FUNCTION_BLOCK MOTOR_TO_EVENTS (* Basic Function Block Type *)
  (* Standard: 61499-2 *)
  (* Version 0.3, 2009-09-15, JHC, Holobloc Inc, Changed transition priorities. *)
  (* Version 0.2, 2003-12-04, JHC, Rockwell Automation, Renamed for better indexing. *)
  (* Version 0.1, 2002-11-05, JHC, Rockwell Automation, Corrected missing ST element in Algorithm REQ. *)
  (* Version 0.0, 2000-05-30, JHC, Rockwell Automation *)
  PACKAGE fb.rt.Conveyer;
  IMPORT fb.datatype.*;
  IMPORT fb.rt.*;
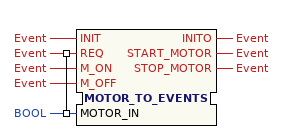
  EVENT_INPUT
    INIT; (* Initialization Request *)
    REQ WITH MOTOR_IN; (* Normal Execution Request *)
    M_ON;
    M_OFF;
  END_EVENT
  EVENT_OUTPUT
    INITO; (* Initialization Confirm *)
    START_MOTOR;
    STOP_MOTOR;
  END_EVENT
  VAR_INPUT
    MOTOR_IN : BOOL;
  END_VAR
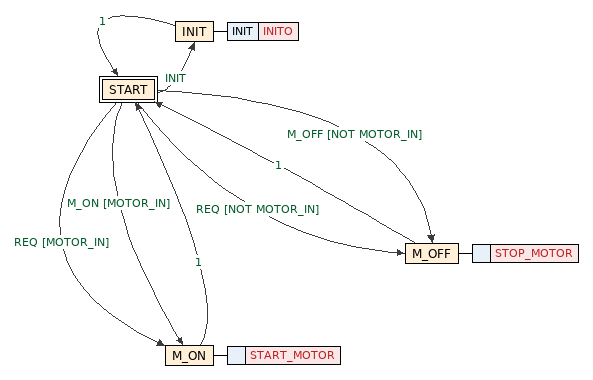
  EC_STATES
    START; (* Initial State *)
    INIT : INIT -> INITO; (* Initialization *)
    M_ON : -> START_MOTOR;
    M_OFF : -> STOP_MOTOR;
  END_STATES
  EC_TRANSITIONS
    INIT TO START := 1;
    START TO INIT := INIT;
    START TO M_ON := REQ [MOTOR_IN];
    M_ON TO START := 1;
    START TO M_OFF := REQ [NOT MOTOR_IN];
    M_OFF TO START := 1;
    START TO M_ON := M_ON [MOTOR_IN];
    START TO M_OFF := M_OFF [NOT MOTOR_IN];
  END_TRANSITIONS
  ALGORITHM INIT IN ST: (* Initialization algorithm *)

  END_ALGORITHM
END_FUNCTION_BLOCK
